{attribute 'GeneratedUsingTerminal: EL3351-0000-0016'}
{attribute addProperty BoxType "EL3351-0000-0016"}
{attribute addProperty Description "EL3351 1Ch. Ana. Input Resistor Bridge Terminal, Diff. 16bit "}
{attribute addProperty Physics "KK"}
{attribute addProperty Id "AIBridge_InputsAT %I*AIBridge_Inputs_555AA1E89AISupply_InputsAT %I*AISupply_Inputs_555AA1E89WcStateAT %I*WcState_9091E0EB2InfoDataAT %I*InfoData_32EB74EA10"}
{attribute addProperty CRC "1749545603"}
{attribute addProperty Size "30"}
TYPE EL3351_6847F283 EXTENDS EtcSlaveTerminalBase_947E5A46 :
STRUCT
	{attribute addProperty Name "AIBridge_Inputs"}
	AIBridge_Inputs : AIBridge_Inputs_555AA1E8;
	{attribute addProperty Name "AISupply_Inputs"}
	AISupply_Inputs : AISupply_Inputs_555AA1E8;
	{attribute addProperty Name "WcState"}
	WcState : WcState_9091E0EB;
	{attribute addProperty Name "InfoData"}
	InfoData : InfoData_32EB74EA;
END_STRUCT
END_TYPE

(* stored: Version 1.2.0.0, ProductVersion 3.1.4024.9
   DUT EL3351_6847F283: Id {9d66fe63-94ac-439c-b5e2-d416a12ad800} *)
